GLOBALCONSTANTS DefaultPool_PI (* Global constants *)
  PACKAGE Uebungen::const::UT::PI;
  VAR_GLOBAL CONSTANT
    ISO_DESIGNATOR_WIDTH : UINT := 80;
    ISO_DESIGNATOR_HEIGHT : UINT := 80;
    ISO_MASK_SIZE : UINT := 480;
    ISO_VERSION_LABEL : STRING;
    MASK_WIDTH : UINT := 480;
    MASK_HEIGHT : UINT := 480;
    WorkingSet : UINT := 0;
    Macro_M1 : UINT := 1;
    Macro_PI_1 : UINT := 2;
    Macro_PI_2 : UINT := 3;
    Macro_PI_3 : UINT := 4;
    Macro_PI_4 : UINT := 5;
    DataMask_M1 : UINT := 1000;
    DataMask_PI1 : UINT := 1001;
    DataMask_PI2 : UINT := 1002;
    DataMask_PI3 : UINT := 1003;
    DataMask_PI4 : UINT := 1004;
    Container_Q : UINT := 3000;
    SoftKeyMask_PI : UINT := 4000;
    SoftKey_Ausgaenge : UINT := 5000;
    SoftKey_PI1 : UINT := 5001;
    SoftKey_PI2 : UINT := 5002;
    SoftKey_PI3 : UINT := 5003;
    SoftKey_PI4 : UINT := 5004;
    Button_Q01 : UINT := 6001;
    Button_Q02 : UINT := 6002;
    Button_Q03 : UINT := 6003;
    Button_Q04 : UINT := 6004;
    Button_Q05 : UINT := 6005;
    Button_Q06 : UINT := 6006;
    Button_Q07 : UINT := 6007;
    Button_Q08 : UINT := 6008;
    Button_Q09 : UINT := 6009;
    Button_Q10 : UINT := 6010;
    Button_Q11 : UINT := 6011;
    Button_Q12 : UINT := 6012;
    Button_PI_I01_SWITCH : UINT := 6101;
    Button_PI_I01_STATUS : UINT := 6102;
    Button_PI_I02_SWITCH : UINT := 6103;
    Button_PI_I02_STATUS : UINT := 6104;
    Button_PI_I03_SWITCH : UINT := 6105;
    Button_PI_I03_STATUS : UINT := 6106;
    Button_PI_I04_SWITCH : UINT := 6107;
    Button_PI_I04_STATUS : UINT := 6108;
    Button_PI_I05_SWITCH : UINT := 6109;
    Button_PI_I05_STATUS : UINT := 6110;
    Button_PI_I06_SWITCH : UINT := 6111;
    Button_PI_I06_STATUS : UINT := 6112;
    Button_PI_I07_SWITCH : UINT := 6113;
    Button_PI_I07_STATUS : UINT := 6114;
    Button_PI_I08_SWITCH : UINT := 6115;
    Button_PI_I08_STATUS : UINT := 6116;
    OutputString_WorkingSet_0 : UINT := 11000;
    Label_SoftKey_Ausgaenge : UINT := 11001;
    Label_SoftKey_PI1 : UINT := 11002;
    Label_SoftKey_PI2 : UINT := 11003;
    Label_SoftKey_PI3 : UINT := 11004;
    Label_SoftKey_PI4 : UINT := 11005;
    Label_PI_I01 : UINT := 11006;
    Label_PI_I02 : UINT := 11007;
    Label_PI_I03 : UINT := 11008;
    Label_PI_I04 : UINT := 11009;
    Label_PI_I05 : UINT := 11010;
    Label_PI_I06 : UINT := 11011;
    Label_PI_I07 : UINT := 11012;
    Label_PI_I08 : UINT := 11013;
    Label_Btn_SWITCH : UINT := 11014;
    OutputNumber_c1 : UINT := 12001;
    OutputNumber_c9 : UINT := 12009;
    OutputNumber_c10 : UINT := 12010;
    OutputNumber_c11 : UINT := 12011;
    OutputNumber_c12 : UINT := 12012;
    OutputNumber_c2 : UINT := 12013;
    OutputNumber_c3 : UINT := 12014;
    OutputNumber_c4 : UINT := 12015;
    OutputNumber_c5 : UINT := 12016;
    OutputNumber_c6 : UINT := 12017;
    OutputNumber_c7 : UINT := 12018;
    OutputNumber_c8 : UINT := 12019;
    OutputNumber_Tick : UINT := 12020;
    OutputNumber_PI_I01_FREQ : UINT := 12021;
    OutputNumber_PI_I01_COUNT : UINT := 12022;
    OutputNumber_PI_I02_FREQ : UINT := 12023;
    OutputNumber_PI_I02_COUNT : UINT := 12024;
    OutputNumber_PI_I03_FREQ : UINT := 12025;
    OutputNumber_PI_I03_COUNT : UINT := 12026;
    OutputNumber_PI_I04_FREQ : UINT := 12027;
    OutputNumber_PI_I04_COUNT : UINT := 12028;
    OutputNumber_PI_I05_FREQ : UINT := 12029;
    OutputNumber_PI_I05_COUNT : UINT := 12030;
    OutputNumber_PI_I06_FREQ : UINT := 12031;
    OutputNumber_PI_I06_COUNT : UINT := 12032;
    OutputNumber_PI_I07_FREQ : UINT := 12033;
    OutputNumber_PI_I07_COUNT : UINT := 12034;
    OutputNumber_PI_I08_FREQ : UINT := 12035;
    OutputNumber_PI_I08_COUNT : UINT := 12036;
    Bargraph_PI_I01 : UINT := 18000;
    Bargraph_PI_I02 : UINT := 18001;
    Bargraph_PI_I03 : UINT := 18002;
    Bargraph_PI_I04 : UINT := 18003;
    Bargraph_PI_I05 : UINT := 18004;
    Bargraph_PI_I06 : UINT := 18005;
    Bargraph_PI_I07 : UINT := 18006;
    Bargraph_PI_I08 : UINT := 18007;
    Logos_icon : UINT := 20500;
    NumberVariable_PI_FREQ_I01 : UINT := 21000;
    NumberVariable_PI_FREQ_I02 : UINT := 21001;
    NumberVariable_PI_FREQ_I03 : UINT := 21002;
    NumberVariable_PI_FREQ_I04 : UINT := 21003;
    NumberVariable_PI_FREQ_I05 : UINT := 21004;
    NumberVariable_PI_FREQ_I06 : UINT := 21005;
    NumberVariable_PI_FREQ_I07 : UINT := 21006;
    NumberVariable_PI_FREQ_I08 : UINT := 21007;
    NumberVariable_PI_COUNT_I01 : UINT := 21008;
    NumberVariable_PI_COUNT_I02 : UINT := 21009;
    NumberVariable_PI_COUNT_I03 : UINT := 21010;
    NumberVariable_PI_COUNT_I04 : UINT := 21011;
    NumberVariable_PI_COUNT_I05 : UINT := 21012;
    NumberVariable_PI_COUNT_I06 : UINT := 21013;
    NumberVariable_PI_COUNT_I07 : UINT := 21014;
    NumberVariable_PI_COUNT_I08 : UINT := 21015;
    FontAttributes_6x8 : UINT := 23000;
    FontAttributes_24x32 : UINT := 23001;
    FontAttributes_16x16 : UINT := 23002;
    AuxFunction2_X1 : UINT := 31000;
  END_VAR
END_GLOBALCONSTANTS
